// TwinCAT 3 PLC project XtsTransport
// Title: XTS Transport
// Author: D.Hauer
// ProjectVersion: 0.0.1
// Description: basic functionblocks for building XTS transport
// ProgramVersion: 3.1.4024.0
// libraries:
//   Tc2_Math, * (Beckhoff Automation GmbH)
//   Tc2_MC2, * (Beckhoff Automation GmbH)
//   Tc2_Standard, * (Beckhoff Automation GmbH)
//   Tc2_System, * (Beckhoff Automation GmbH)
//   Tc2_Utilities, * (Beckhoff Automation GmbH)
//   Tc3_McCollisionAvoidance, * (Beckhoff Automation GmbH)
//   Tc3_McCoordinatedMotion, * (Beckhoff Automation GmbH)
//   Tc3_Module, * (Beckhoff Automation GmbH)
//   Tc3_XTS_Utility, * (Beckhoff Automation GmbH)
//   VisuDialogs, * (System)
// project tree:
//   DUTs/_Visu/ ST_VisuExampleIO.TcDUT
//   / GlobalTextList.TcGTLO (not stored), MAIN.TcPOU (not stored), PlcTask.TcTTO (not stored), Visualization Manager.TcVMO (not stored)
//   POUs/ FB_OperatingMode.TcPOU, FB_SimpleCaExample.TcPOU (not stored)
//   VISUs/ CA_Visu.TcVIS
//   VISUs/Frame/ FrameVisuSimpelCaExample.TcVIS
//   VISUs/Frame/SubFrame/ FrameAdvancedMotion.TcVIS, FrameDummy.TcVIS, FrameXtsStateModel.TcVIS, FrameDislaimer.TcVIS
//   XTS/CaGroup/ FB_CaGroup.TcPOU, I_CaGroup.TcIO (not stored)
//   XTS/CaGroup/old/ fb_CaGroup_withOutInterface.TcPOU (not stored), fb_GroupCtrl.TcPOU
//   XTS/CaGroup/types/ E_GROUP_CHECK.TcDUT (not stored), E_GROUP_CTRL.TcDUT, E_GROUP_STATE.TcDUT, ST_GROUP_CTRL.TcDUT (not stored), ST_GROUP_INFO.TcDUT (not stored), ST_GROUP_STATE.TcDUT
//   XTS/ GVL_XTS.TcGVL (not stored), Param.TcGVL
//   XTS/Mover/ fb_Mover.TcPOU (not stored), I_Mover.TcIO, I_StationMover.TcIO
//   XTS/Mover/old/ fb_MoverCtrl.TcPOU (not stored), fb_Mover_withOutInterface.TcPOU (not stored)
//   XTS/Mover/types/ E_MOVER_CTRL.TcDUT (not stored), E_MOVER_STATE.TcDUT (not stored), ST_GEAR_DATA.TcDUT (not stored), ST_MOVER_CTRL.TcDUT (not stored), ST_MOVER_INFO.TcDUT (not stored), ST_MOVER_STATE.TcDUT (not stored), ST_MOVE_DATA.TcDUT (not stored)
//   XTS/Station/ fb_Station.TcPOU (not stored)
//   XTS/Station/types/ E_STATION_CTRL.TcDUT (not stored), E_STATION_STATE.TcDUT, fb_Station_LinkedListCtrl.TcPOU (not stored), I_Station_LinkedList.TcIO, ST_STATION_CTRL.TcDUT (not stored), ST_STATION_LIST_RESULT.TcDUT (not stored), ST_STATION_MOVER_DATA.TcDUT, ST_STATION_PARAMETER.TcDUT (not stored), ST_STATION_STATE.TcDUT, T_NEST_OFFSET.TcDUT
//   XTS/_types/ E_OperatingState.TcDUT (not stored), E_OperatingCmd.TcDUT (not stored), E_PROGRESS.TcDUT (not stored)

// ---- DUTs/_Visu/ST_VisuExampleIO.TcDUT
TYPE ST_VisuExampleIO :
STRUCT
	
	bStart				: BOOL;
	iState				: INT;
	bAgain				: BOOL := TRUE;
	fSetPos1			: LREAL := 1000;
	fSetPos2			: LREAL := 1250;
	fSetPos3			: LREAL := 1990;

	bStepModeActive		: BOOL;
	bNextStep			: BOOL;
	
// Operatin State
	eOPMState			: E_OperatingState;
	eLastOPMState		: E_OperatingState;
	eStateCommand		: E_OperatingCmd;
	
// CaGroup State
	stCaGroup			: REFERENCE TO AXES_GROUP_REF;	
	
END_STRUCT
END_TYPE

// ---- XTS/CaGroup/types/E_GROUP_CTRL.TcDUT
{attribute 'qualified_only'}
{attribute 'strict'}
{attribute 'to_string'}
TYPE E_GROUP_CTRL :
(
  GROUP_INVALID,
  GROUP_INIT    := 10,
  GROUP_CLEAR,
  GROUP_BUILD,
  GROUP_ENABLE
)UINT;
END_TYPE

// ---- XTS/CaGroup/types/E_GROUP_STATE.TcDUT
{attribute 'qualified_only'}
{attribute 'to_string'}
TYPE E_GROUP_STATE :
(
  GROUP_INVALID,
  GROUP_INIT    := 10,
  GROUP_CLEAR,
  GROUP_BUILD,
  GROUP_ENABLE

)UINT;
END_TYPE

// ---- XTS/CaGroup/types/ST_GROUP_STATE.TcDUT
TYPE ST_GROUP_STATE :
STRUCT
  State           : E_GROUP_STATE;
  McState         : MC_GROUP_STATE;
  AxisCount       : UINT;
END_STRUCT
END_TYPE

// ---- XTS/Station/types/E_STATION_STATE.TcDUT
{attribute 'to_string'}
TYPE E_STATION_STATE :
(
	STATION_NO_INIT,                // startup state after power on
  STATION_INIT,                   // station and list/queue cleared;
  STATION_DISABLE         := 10,  // check enable from ctrl
  STATION_ENABLE,                 // check enable from ctrl
  STATION_DETECT_MOVER,           // wait until queue > 0
  STATION_MOVER_ENTER     := 20,  // mover asking for entry
  STATION_MOVER_IN_TARGET,        // mover moving to PosWork
  STATION_PROCESS_START   := 30,  // wait until process started
  STATION_PROCESS_DONE,           // wait until process done
  STATION_CHECK           := 40,  // check for next nest in mask
  STATION_CHECK_NEST,             // get next nest position
  STATION_MOVER_OUT       := 50,  // mover asking to leave
  STATION_MOVER_RELEASE,          // check if release distance is passed
  STATION_MOVER_GONE,             // mover out of station, enter mover in target station list


  STATION_ERROR           := 127,
  STATION_ERROR_LIST_GET_HEAD_FAULT,
  STATION_ERROR_LIST_REMOVE_HEAD_FAULT,
  STATION_ERROR_LIST_ADD_TAIL_FAULT,
  STATION_ERROR_LIST_STATION_ID_WRONG,
  STATION_ERROR_LIST_MOVER_ID_INVALID,
  STATION_ERROR_INFEED_ERROR,
  STATION_ERROR_OUTFEED_TARGET_INVALID,

  STATION_ERROR_FATAL     := 255 // the thing that must not be
)USINT;
END_TYPE

// ---- XTS/Station/types/ST_STATION_MOVER_DATA.TcDUT
{attribute 'pack_mode' := '2'}
TYPE ST_STATION_MOVER_DATA :
STRUCT
  nMoverId        : USINT;  // who am I?  !! MUST be correct !! - movement to base position sets everything in order, DO NOT manipulate!
  nTargetStation  : USINT;  // where shall I be? used for double checking with StationId at infeed of mover into station

  {attribute 'displaymode':='bin'}
  nMask           : BYTE;   // how many of you are there? (1 = default, no action required)

  rOffset         : REAL;   // offset for use in work flow !! added to static mover offset for every nest(bit) in nMask!!
END_STRUCT
END_TYPE

// ---- XTS/Station/types/ST_STATION_STATE.TcDUT
{attribute 'pack_mode' := '2'}
TYPE ST_STATION_STATE :
STRUCT
  eState          : E_STATION_STATE;
  {attribute 'displaymode':='bin'}
  nMask           : BYTE;
  nMoverId        : USINT;
  nQueue          : USINT; // queue count for station
END_STRUCT
END_TYPE

// ---- XTS/Station/types/T_NEST_OFFSET.TcDUT
TYPE T_NEST_OFFSET : ARRAY[1..MAX_MOVER]        OF
                     ARRAY[1..MAX_STATION_POS]  OF LREAL;
END_TYPE

// ---- XTS/Param.TcGVL
//{attribute 'qualified_only'}
VAR_GLOBAL CONSTANT
// HAUD 2023 12 13
  Version             : STRING  := '3.2.0'; // V3.2.0 - design test with references, improved separation of Mover and Group handling, redesign of group handling



// XTS-Constant ´--> using Tc3_XTS_Utility.TcIoXtsEnvironmentParameterList


  MAX_INFO_SERVER     : UINT    :=  TO_UINT(Tc3_XTS_Utility.TcIoXtsEnvironmentParameterList.MaxXtsInfoServer);
  MAX_INFO_STATION    : UINT    :=  TO_UINT(Tc3_XTS_Utility.TcIoXtsEnvironmentParameterList.MaxXtsInfoStation);
  MAX_INFO_STOP_POS   : UINT    :=  TO_UINT(Tc3_XTS_Utility.TcIoXtsEnvironmentParameterList.MaxXtsStopPositionsPerStation);


  MAX_MOVER           : UINT    := TO_UINT(Tc3_XTS_Utility.TcIoXtsEnvironmentParameterList.MaxXtsMoversPerXpu);
  MAX_MODULE          : UINT    := TO_UINT(Tc3_XTS_Utility.TcIoXtsEnvironmentParameterList.MaxModulesPerPart);
  MAX_PART            : UINT    := TO_UINT(Tc3_XTS_Utility.TcIoXtsEnvironmentParameterList.MaxXtsPartsPerXpu);
  MAX_TRACK           : UINT    := TO_UINT(Tc3_XTS_Utility.TcIoXtsEnvironmentParameterList.MaxXtsTracksPerXpu);
  MAX_GROUP           : UINT    := TO_UINT(Tc3_XTS_Utility.TcIoXtsEnvironmentParameterList.MaxXtsCaGroup);

  MAX_STATION         : UINT    := 2;
  MAX_STATION_POS     : UINT    := TO_UINT(SIZEOF(ST_STATION_STATE.nMask)*8);
  MAX_LIST_NODES      : UINT    := MAX_MOVER;
  MAX_MASTER          : UINT    := 1;
  
END_VAR

// ---- XTS/Mover/I_Mover.TcIO
INTERFACE I_Mover

METHOD Disable : E_PROGRESS
VAR_INPUT
  Execute             : BOOL;
END_VAR
END_METHOD

METHOD Enable : E_PROGRESS
VAR_INPUT
  Execute             : BOOL;
END_VAR
END_METHOD

METHOD GearIn : E_PROGRESS;
VAR_INPUT
  Execute             : BOOL;
  stGearData          : ST_GEAR_DATA;
  stMoveData          : ST_MOVE_DATA;
END_VAR
END_METHOD

METHOD GearInPosCa : E_PROGRESS
VAR_INPUT
  Execute             : BOOL;
  stMoveData          : ST_MOVE_DATA;
  stGearData          : ST_GEAR_DATA;  
END_VAR
END_METHOD

METHOD GearOut : E_PROGRESS
VAR_INPUT
  Execute             : BOOL;
END_VAR
END_METHOD

METHOD GetMoverInfo : ST_MOVER_INFO
VAR_INPUT
END_VAR
END_METHOD

METHOD Halt : E_PROGRESS
VAR_INPUT
  Execute             : BOOL;
  stMoveData          : ST_MOVE_DATA;
END_VAR
END_METHOD

PROPERTY LastGap : REFERENCE to lreal
SET
END_SET
END_PROPERTY

PROPERTY LastPosition : REFERENCE to LREAL
SET
END_SET
END_PROPERTY

PROPERTY Master : REFERENCE to AXIS_REF
SET
END_SET
END_PROPERTY

PROPERTY Mover : REFERENCE to AXIS_REF
SET
END_SET
END_PROPERTY

METHOD MoveToPosCa : E_PROGRESS
VAR_INPUT
  Execute             : BOOL;
  stMoveData          : ST_MOVE_DATA;
END_VAR
END_METHOD

PROPERTY RailLength : LREAL
GET
END_GET
SET
END_SET
END_PROPERTY

METHOD Reset : E_PROGRESS
VAR_INPUT
  Execute             : BOOL;
END_VAR
END_METHOD

METHOD SendToPosCa : E_PROGRESS
VAR_INPUT
  Execute             : BOOL;
  stMoveData          : ST_MOVE_DATA;
END_VAR
END_METHOD

END_INTERFACE

// ---- XTS/Mover/I_StationMover.TcIO
INTERFACE I_StationMover

METHOD GetMoverInfo : ST_MOVER_INFO
VAR_INPUT
END_VAR
END_METHOD

METHOD MoveToPosCa : E_PROGRESS
VAR_INPUT
  Execute             : BOOL;
  stMoveData          : ST_MOVE_DATA;
END_VAR
END_METHOD

PROPERTY RailLength : LREAL
GET
END_GET
END_PROPERTY

METHOD SendToPosCa : E_PROGRESS
VAR_INPUT
  Execute             : BOOL;
  stMoveData          : ST_MOVE_DATA;
END_VAR
END_METHOD

END_INTERFACE

// ---- XTS/Station/types/I_Station_LinkedList.TcIO
INTERFACE I_Station_LinkedList

METHOD AddHeadValue : ST_STATION_LIST_RESULT
VAR_INPUT
  stData        : ST_STATION_MOVER_DATA;
END_VAR
END_METHOD

METHOD AddTailValue : ST_STATION_LIST_RESULT
VAR_INPUT
  stData          : ST_STATION_MOVER_DATA;
END_VAR
END_METHOD

PROPERTY Count : UDINT
GET
END_GET
END_PROPERTY

PROPERTY Data : ARRAY[0..MAX_LIST_NODES] OF ST_STATION_MOVER_DATA
GET
END_GET
END_PROPERTY

PROPERTY Free : UDINT
GET
END_GET
END_PROPERTY

METHOD GetHead : ST_STATION_LIST_RESULT
VAR_INPUT
END_VAR
END_METHOD

METHOD InitList : BOOL
END_METHOD

PROPERTY Nodes : ARRAY[0..MAX_LIST_NODES] OF T_LinkedListEntry
GET
END_GET
END_PROPERTY

METHOD RemoveHeadValue : ST_STATION_LIST_RESULT
VAR_INPUT
END_VAR
END_METHOD

END_INTERFACE

// ---- POUs/FB_OperatingMode.TcPOU
FUNCTION_BLOCK FB_OperatingMode
//---------------------------------------------------------------------------------------------------------------
//
//  Fen 2023.12.21
//
//  - XTS_TRAINING
//  - example project for setting up transport layer
//
//
//  FB_OperatingMode
//  - Operating Mode handler for XTS_training Exsample
//  - 
//
//
//---------------------------------------------------------------------------------------------------------------
// This SOFTWARE is provided as an Exemple by THE PROVIDER "as is" and "with all faults." THE PROVIDER makes no 
// representations or warranties of any kind concerning the safety, suitability, lack of viruses, inaccuracies, 
// typographical errors, or other harmful components of this SOFTWARE. There are inherent dangers in the use of 
// any software, and you are solely responsible for determining whether this SOFTWARE is compatible with your 
// equipment and other software installed on your equipment. You are also solely responsible for the protection 
// of your equipment and backup of your data, and THE PROVIDER will not be liable for any damages you may suffer 
// in connection with using, modifying, or distributing this SOFTWARE.
//---------------------------------------------------------------------------------------------------------------

VAR 
	_eState			: E_OperatingState;	
	_eLastState		: E_OperatingState;

	_eCommand		: E_OperatingCmd;
	_eActCommand	: E_OperatingCmd;
	

	_StaeCompleteRtrig	:R_TRIG;
	_StaeComplete		: BOOL;

	
	_bSingelStep				: BOOL;

END_VAR

PROPERTY Command : E_OperatingCmd
GET

	Command := _eActCommand;
END_GET
SET

	_eCommand := Command;
END_SET
END_PROPERTY

METHOD Cyclic
VAR_INPUT
END_VAR
// simple Example for Operatingmode handler


// State Complete
	_StaeCompleteRtrig();
	IF _StaeCompleteRtrig.Q THEN
		_StaeComplete := TRUE;
	END_IF

// Xts Operating Mode

	_eActCommand := _eActCommand;

	CASE _eState OF
	
	// Invalid 	--> wait for Cmd 	
	E_OperatingState.OperatingMode_INVALID : 
		IF _eCommand = E_OperatingCmd.OperatingCmd_Clear THEN
			_eState := E_OperatingState.OperatingMode_Clear;
			_eActCommand := E_OperatingCmd.OperatingCmd_DONE;
			_eLastState := E_OperatingState.OperatingMode_INVALID;
		
		ELSE 
			_eActCommand := E_OperatingCmd.OperatingCmd_DONE;	
		END_IF
		
	// Clear 	--> Init Ca-Group  and Axis 	
	E_OperatingState.OperatingMode_Clear:
		IF _StaeComplete 
		THEN
			_StaeComplete := FALSE;
			_eState := E_OperatingState.OperatingMode_Clear_Sc;
		END_IF
		
		CASE _eCommand	OF  			
			E_OperatingCmd.OperatingCmd_Reset :	
				_eState := E_OperatingState.OperatingMode_Reset;
				_eActCommand := E_OperatingCmd.OperatingCmd_DONE;
				_eLastState := E_OperatingState.OperatingMode_Clear;
			
		ELSE 
			_eActCommand := E_OperatingCmd.OperatingCmd_DONE;	
				
		END_CASE
		
	// Clear_Sc 	--> State complete	
	E_OperatingState.OperatingMode_Clear_Sc :
		CASE _eCommand	OF  
			E_OperatingCmd.OperatingCmd_Clear :
				_eState := E_OperatingState.OperatingMode_Clear;
				_eActCommand := E_OperatingCmd.OperatingCmd_DONE;
				_eLastState := E_OperatingState.OperatingMode_Clear_Sc;
			
			E_OperatingCmd.OperatingCmd_Reset :	
				_eState := E_OperatingState.OperatingMode_Reset;
				_eActCommand := E_OperatingCmd.OperatingCmd_DONE;
				_eLastState := E_OperatingState.OperatingMode_Clear_Sc;
				
			E_OperatingCmd.OperatingCmd_Prepare	:
				_eState := E_OperatingState.OperatingMode_Prepare;
				_eActCommand := E_OperatingCmd.OperatingCmd_DONE;
				_eLastState := E_OperatingState.OperatingMode_Clear_Sc;
		
		ELSE 
			_eActCommand := E_OperatingCmd.OperatingCmd_DONE;	
				
		END_CASE
		
	
	// Prepare 	--> build Ca-Group  and enable Axis 	
	E_OperatingState.OperatingMode_Prepare :
		IF _StaeComplete 
		THEN
			_StaeComplete := FALSE;
			_eState := E_OperatingState.OperatingMode_Prepar_Sc;
		END_IF
		
		CASE _eCommand	OF  
			E_OperatingCmd.OperatingCmd_Clear :
				_eState := E_OperatingState.OperatingMode_Clear;
				_eActCommand := E_OperatingCmd.OperatingCmd_DONE;
				_eLastState := E_OperatingState.OperatingMode_Prepare;
			
			E_OperatingCmd.OperatingCmd_Reset :	
				_eState := E_OperatingState.OperatingMode_Reset;
				_eActCommand := E_OperatingCmd.OperatingCmd_DONE;
				_eLastState := E_OperatingState.OperatingMode_Prepare;
		
		ELSE 
			_eActCommand := E_OperatingCmd.OperatingCmd_DONE;	
		END_CASE
	
	// Stopping 	--> stop Axis 		
	E_OperatingState.OperatingMode_Stopping :
		IF _StaeComplete 
		THEN
			_StaeComplete := FALSE;
			_eState := E_OperatingState.OperatingMode_Prepar_Sc;
		END_IF
		CASE _eCommand	OF  
			E_OperatingCmd.OperatingCmd_Clear :
				_eState := E_OperatingState.OperatingMode_Clear;
				_eActCommand := E_OperatingCmd.OperatingCmd_DONE;
				_eLastState := E_OperatingState.OperatingMode_Stopping;
			
			E_OperatingCmd.OperatingCmd_Reset :	
				_eState := E_OperatingState.OperatingMode_Reset;
				_eActCommand := E_OperatingCmd.OperatingCmd_DONE;
				_eLastState := E_OperatingState.OperatingMode_Stopping;
		
		ELSE 
			_eActCommand := E_OperatingCmd.OperatingCmd_DONE;	
		END_CASE
		
	// Prepare 	--> emptying the system 		
	E_OperatingState.OperatingMode_Empty:
		IF _StaeComplete 
		THEN
			_StaeComplete := FALSE;
			_eState := E_OperatingState.OperatingMode_Prepar_Sc;
		END_IF
		
		CASE _eCommand	OF  
			E_OperatingCmd.OperatingCmd_Clear :
				_eState := E_OperatingState.OperatingMode_Clear;
				_eActCommand := E_OperatingCmd.OperatingCmd_DONE;
				_eLastState := E_OperatingState.OperatingMode_Empty;
			
			E_OperatingCmd.OperatingCmd_Reset :	
				_eState := E_OperatingState.OperatingMode_Reset;
				_eActCommand := E_OperatingCmd.OperatingCmd_DONE;
				_eLastState := E_OperatingState.OperatingMode_Empty;
				
			E_OperatingCmd.OperatingCmd_Stopping :
				_eState := E_OperatingState.OperatingMode_Stopping;
				_eActCommand := E_OperatingCmd.OperatingCmd_DONE;
				_eLastState := E_OperatingState.OperatingMode_Empty;
		
		ELSE 
			_eActCommand := E_OperatingCmd.OperatingCmd_DONE;	
			
		END_CASE
	
	// 	Prepare 	--> State complete
	E_OperatingState.OperatingMode_Prepar_Sc:
		CASE _eCommand	OF  
			E_OperatingCmd.OperatingCmd_Clear :
				_eState := E_OperatingState.OperatingMode_Clear;
				_eActCommand := E_OperatingCmd.OperatingCmd_DONE;
				_eLastState := E_OperatingState.OperatingMode_Prepar_Sc;
			
			E_OperatingCmd.OperatingCmd_Reset :	
				_eState := E_OperatingState.OperatingMode_Reset;
				_eActCommand := E_OperatingCmd.OperatingCmd_DONE;
				_eLastState := E_OperatingState.OperatingMode_Prepar_Sc;
				
			E_OperatingCmd.OperatingCmd_Stopping :
				_eState := E_OperatingState.OperatingMode_Stopping;
				_eActCommand := E_OperatingCmd.OperatingCmd_DONE;
				_eLastState := E_OperatingState.OperatingMode_Prepar_Sc;
			
			E_OperatingCmd.OperatingCmd_Home 	:
				_eState := E_OperatingState.OperatingMode_Home;
				_eActCommand := E_OperatingCmd.OperatingCmd_DONE;
				_eLastState := E_OperatingState.OperatingMode_Prepar_Sc;
		
		ELSE 
			_eActCommand := E_OperatingCmd.OperatingCmd_DONE;	
	
		END_CASE
		
	// 	Empty 	--> State complete
	E_OperatingState.OperatingMode_Empty_Sc:
			_eState := E_OperatingState.OperatingMode_Prepar_Sc;
			_eLastState := E_OperatingState.OperatingMode_Empty_Sc;
		
	// 	Stopping 	--> State complete
	E_OperatingState.OperatingMode_Stopping_Sc:
			_eState := E_OperatingState.OperatingMode_Prepar_Sc;
			_eLastState := E_OperatingState.OperatingMode_Stopping_Sc;


	
	// 	Home 	--> Move to Start Position
	E_OperatingState.OperatingMode_Home :
		IF _StaeComplete 
		THEN
			_StaeComplete := FALSE;
			_eState := E_OperatingState.OperatingMode_Home_Sc;
		END_IF
		
		CASE _eCommand	OF  
			E_OperatingCmd.OperatingCmd_Clear :
				_eState := E_OperatingState.OperatingMode_Clear;
				_eActCommand := E_OperatingCmd.OperatingCmd_DONE;
				_eLastState := E_OperatingState.OperatingMode_Home;
			
			E_OperatingCmd.OperatingCmd_Reset :	
				_eState := E_OperatingState.OperatingMode_Reset;
				_eActCommand := E_OperatingCmd.OperatingCmd_DONE;
				_eLastState := E_OperatingState.OperatingMode_Home;
				
			E_OperatingCmd.OperatingCmd_Stopping :
				_eState := E_OperatingState.OperatingMode_Stopping;
				_eActCommand := E_OperatingCmd.OperatingCmd_DONE;
				_eLastState := E_OperatingState.OperatingMode_Home;
		
		ELSE 
			_eActCommand := E_OperatingCmd.OperatingCmd_DONE;	
	
		END_CASE
	
	// 	Home 	--> State complete
	E_OperatingState.OperatingMode_Home_Sc :	
		_eState := E_OperatingState.OperatingMode_Active;
		
		CASE _eCommand	OF  
			E_OperatingCmd.OperatingCmd_Clear :
				_eState := E_OperatingState.OperatingMode_Clear;
				_eActCommand := E_OperatingCmd.OperatingCmd_DONE;
				_eLastState := E_OperatingState.OperatingMode_Home_Sc;
			
			E_OperatingCmd.OperatingCmd_Reset :	
				_eState := E_OperatingState.OperatingMode_Reset;
				_eActCommand := E_OperatingCmd.OperatingCmd_DONE;
				_eLastState := E_OperatingState.OperatingMode_Home_Sc;
				
			E_OperatingCmd.OperatingCmd_Stopping :
				_eState := E_OperatingState.OperatingMode_Stopping;
				_eActCommand := E_OperatingCmd.OperatingCmd_DONE;
				_eLastState := E_OperatingState.OperatingMode_Home_Sc;
		
		ELSE 
			_eActCommand := E_OperatingCmd.OperatingCmd_DONE;	
	
		END_CASE
	
	// 	Active/Work 	--> execute work sequences
 	E_OperatingState.OperatingMode_Active :
		CASE _eCommand	OF  
			E_OperatingCmd.OperatingCmd_Clear :
				_eState := E_OperatingState.OperatingMode_Clear;
				_eActCommand := E_OperatingCmd.OperatingCmd_DONE;
				_eLastState := E_OperatingState.OperatingMode_Active;
			
			E_OperatingCmd.OperatingCmd_Reset :	
				_eState := E_OperatingState.OperatingMode_Reset;
				_eActCommand := E_OperatingCmd.OperatingCmd_DONE;
				_eLastState := E_OperatingState.OperatingMode_Active;
				
			E_OperatingCmd.OperatingCmd_Stopping :
				_eState := E_OperatingState.OperatingMode_Stopping;
				_eActCommand := E_OperatingCmd.OperatingCmd_DONE;
				_eLastState := E_OperatingState.OperatingMode_Active;
			
			E_OperatingCmd.OperatingCmd_Empty 	:
				_eState := E_OperatingState.OperatingMode_Empty;
				_eActCommand := E_OperatingCmd.OperatingCmd_DONE;
				_eLastState := E_OperatingState.OperatingMode_Active;
		
		ELSE 
			_eActCommand := E_OperatingCmd.OperatingCmd_DONE;	
				
		END_CASE
	
	// 	Reset 	--> Reset Error --> Jump to last state back
	E_OperatingState.OperatingMode_Reset :
		IF _StaeComplete 
		THEN
			_StaeComplete := FALSE;
			_eState := _eLastState;
			_eLastState := E_OperatingState.OperatingMode_Reset;
		END_IF
	
		_eActCommand := E_OperatingCmd.OperatingCmd_DONE;
		
	
	END_CASE
END_METHOD

PROPERTY eLastState : E_OperatingState
GET

	eLastState := _eLastState;
END_GET
END_PROPERTY

PROPERTY eState : E_OperatingState
GET

	eState := _eState;
END_GET
END_PROPERTY

METHOD M_StateComplete
VAR_INPUT
END_VAR

	//_StaeCompleteRtrig.CLK := TRUE;
	_StaeComplete := TRUE;
END_METHOD

PROPERTY sState : STRING
GET

	sState := to_String(_eState);
END_GET
END_PROPERTY

END_FUNCTION_BLOCK

// ---- XTS/CaGroup/FB_CaGroup.TcPOU
//---------------------------------------------------------------------------------------------------------------
//
//  HAUD 2023.12.13
//
//
//  fb_CaGroup
//  - handles CA group states
//  - add mover to group
//  - remove mover from group
//  - clear group error
//  - startup procedure for getting group ready to work
//
//
//  VAR INPUT / OUTPUT --> see properties
//
//---------------------------------------------------------------------------------------------------------------//
// This SOFTWARE is provided as an Exemple by THE PROVIDER "as is" and "with all faults." THE PROVIDER makes no  //
// representations or warranties of any kind concerning the safety, suitability, lack of viruses, inaccuracies,  //
// typographical errors, or other harmful components of this SOFTWARE. There are inherent dangers in the use of  //
// any software, and you are solely responsible for determining whether this SOFTWARE is compatible with your    //
// equipment and other software installed on your equipment. You are also solely responsible for the protection  //
// of your equipment and backup of your data, and THE PROVIDER will not be liable for any damages you may suffer //
// in connection with using, modifying, or distributing this SOFTWARE.                                           //
//---------------------------------------------------------------------------------------------------------------//
FUNCTION_BLOCK FB_CaGroup	IMPLEMENTS I_CaGroup
VAR
  _eCheck                     : E_GROUP_CHECK;
  _bError                     : BOOL;

  _GroupRef                   : REFERENCE TO Tc3_McCoordinatedMotion.AXES_GROUP_REF;
  _GroupCommon                : MCTOPLC_GROUP_COMMON_PART;

  _AxisRefMover               : REFERENCE TO ARRAY[1..MAX_MOVER] OF Tc2_MC2.AXIS_REF;


  // MC2 function block for halting all motion commands on mover before switching off group
  _fbHalt                     : ARRAY[1..MAX_MOVER] OF Tc2_MC2.MC_Halt;
  _fbReset                    : ARRAY[1..MAX_MOVER] OF Tc2_MC2.MC_Reset;

  // CA group fb instances
  _fbAddAxisGroup             : ARRAY[1..MAX_MOVER] OF Tc3_McCoordinatedMotion.MC_AddAxisToGroup;
  _fbRemoveAxisGroup          : ARRAY[1..MAX_MOVER] OF Tc3_McCoordinatedMotion.MC_RemoveAxisFromGroup;

  _fbGroupDisable             : Tc3_McCoordinatedMotion.MC_GroupDisable;
  _fbGroupEnable              : Tc3_McCoordinatedMotion.MC_GroupEnable;
  _fbGroupErrorRead           : Tc3_McCoordinatedMotion.MC_GroupReadError;
  _fbGroupStatusRead          : Tc3_McCoordinatedMotion.MC_GroupReadStatus;
  _fbGroupReset               : Tc3_McCoordinatedMotion.MC_GroupReset;

  _stGroupInfo                : ST_GROUP_INFO;  // additional bits about the state of the CA group

  _rtrigGroupStatusRead,
  _rtrigGroupErrorRead        : Tc2_Standard.R_TRIG;


END_VAR

METHOD AddAll : E_PROGRESS
VAR_INPUT
  Execute     : BOOL;
END_VAR
VAR_INST
  _nErrorId   : UDINT;
  _eState     : E_PROGRESS;

  _nMover     : UINT;
END_VAR
IF NOT Execute THEN _eState     := E_PROGRESS.PROGRESS_INIT; END_IF 
IF NOT Check() THEN AddAll := E_PROGRESS.PROGRESS_ERROR; RETURN; END_IF


CASE _eState
OF
  E_PROGRESS.PROGRESS_INIT:
    IF Execute
    THEN
      _nErrorId               := 0;
      _nMover                 := 1;
      _eState                 := E_PROGRESS.PROGRESS_BUSY;
    END_IF
END_CASE
//-----------------------------------------------------------------------------
//-----------------------------------------------------------------------------
CASE _eState
OF
  E_PROGRESS.PROGRESS_BUSY:
    _eState                   := E_PROGRESS.PROGRESS_PREPARE;
    _fbAddAxisGroup[_nMover](
                AxesGroup     := _GroupRef, 
                Axis          := _AxisRefMover[_nMover], 
                Execute       := FALSE, 
                IdentInGroup  := UDINT_TO_IDENTINGROUP(_AxisRefMover[_nMover].NcToPlc.AxisId));
END_CASE
//-----------------------------------------------------------------------------
//-----------------------------------------------------------------------------
CASE _eState
OF
  E_PROGRESS.PROGRESS_PREPARE:
    _fbAddAxisGroup[_nMover](
                AxesGroup     := _GroupRef, 
                Axis          := _AxisRefMover[_nMover], 
                Execute       := TRUE, 
                IdentInGroup  := UDINT_TO_IDENTINGROUP(_AxisRefMover[_nMover].NcToPlc.AxisId));

    IF (_fbAddAxisGroup[_nMover].Error)
    THEN
      _eState                 := E_PROGRESS.PROGRESS_ERROR;
      _nErrorId               := _fbAddAxisGroup[_nMover].ErrorId;

    ELSIF (_fbAddAxisGroup[_nMover].Done)
    THEN
      _eState                 := E_PROGRESS.PROGRESS_CHECK;
    END_IF
END_CASE
//-----------------------------------------------------------------------------
//-----------------------------------------------------------------------------
CASE _eState
OF
  E_PROGRESS.PROGRESS_CHECK:
    _eState                   := E_PROGRESS.PROGRESS_OCCUPIED;
    _fbAddAxisGroup[_nMover](
                AxesGroup     := _GroupRef, 
                Axis          := _AxisRefMover[_nMover], 
                Execute       := FALSE, 
                IdentInGroup  := UDINT_TO_IDENTINGROUP(_AxisRefMover[_nMover].NcToPlc.AxisId));
END_CASE
//-----------------------------------------------------------------------------
//-----------------------------------------------------------------------------
CASE _eState
OF
  E_PROGRESS.PROGRESS_OCCUPIED:
    _nMover                   := _nMover + 1;

    IF NOT (_nMover > MAX_MOVER)
    THEN
      _eState                 := E_PROGRESS.PROGRESS_BUSY;
    ELSE
      _eState                 := E_PROGRESS.PROGRESS_DONE;
    END_IF
END_CASE
//-----------------------------------------------------------------------------
//-----------------------------------------------------------------------------

AddAll                   := _eState;
END_METHOD

PROPERTY AxisRef : REFERENCE TO ARRAY[1..MAX_MOVER] OF Tc2_MC2.AXIS_REF
SET
_AxisRefMover REF= AxisRef;
END_SET
END_PROPERTY

METHOD PROTECTED Check : BOOL

IF NOT __ISVALIDREF(_GroupRef)
THEN
  _eCheck                     := E_GROUP_CHECK.CHECK_GROUP_REF_INVALID;
  RETURN;
END_IF

IF NOT __ISVALIDREF(_AxisRefMover)
THEN
  _eCheck                     := E_GROUP_CHECK.CHECK_AXIS_REF_INVALID;
  RETURN;
END_IF

_eCheck                       := E_GROUP_CHECK.CHECK_DONE;
Check                         := TRUE;
END_METHOD

METHOD Disable : E_PROGRESS
VAR_INPUT
  Execute     : BOOL;
END_VAR
VAR_INST
  _nErrorId   : UDINT;
  _eState     : E_PROGRESS;

  _nMover     : UINT;
END_VAR
IF NOT Execute THEN _eState       := E_PROGRESS.PROGRESS_INIT; END_IF 
IF NOT Check() THEN Disable  := E_PROGRESS.PROGRESS_ERROR; RETURN; END_IF


CASE _eState
OF
  E_PROGRESS.PROGRESS_INIT:
    IF Execute
    THEN
      _nErrorId               := 0;
      _nMover                 := 1;
      _eState                 := E_PROGRESS.PROGRESS_BUSY;
    END_IF
END_CASE
//-----------------------------------------------------------------------------
//-----------------------------------------------------------------------------
CASE _eState
OF
  E_PROGRESS.PROGRESS_BUSY:
    _eState                   := E_PROGRESS.PROGRESS_PREPARE;
    _fbGroupDisable(
              AxesGroup       := _GroupRef, 
              Execute         := FALSE); 
END_CASE
//-----------------------------------------------------------------------------
//-----------------------------------------------------------------------------
CASE _eState
OF
  E_PROGRESS.PROGRESS_PREPARE:
    _fbGroupDisable(
              AxesGroup       := _GroupRef, 
              Execute         := TRUE); 

    IF (_fbGroupDisable.Error)
    THEN
      _eState                 := E_PROGRESS.PROGRESS_ERROR;
      _nErrorId               := _fbGroupDisable.ErrorId;
      _fbGroupDisable(
              AxesGroup       := _GroupRef, 
              Execute         := FALSE); 


    ELSIF (_fbGroupDisable.Done)
    THEN
      _eState                 := E_PROGRESS.PROGRESS_DONE;
      _fbGroupDisable(
              AxesGroup       := _GroupRef, 
              Execute         := FALSE); 
    END_IF
END_CASE
//-----------------------------------------------------------------------------
//-----------------------------------------------------------------------------

Disable                  := _eState;
END_METHOD

METHOD Enable : E_PROGRESS
VAR_INPUT
  Execute     : BOOL;
END_VAR
VAR_INST
  _nErrorId   : UDINT;
  _eState     : E_PROGRESS;

  _nMover     : UINT;
END_VAR
IF NOT Execute THEN _eState       := E_PROGRESS.PROGRESS_INIT; END_IF 
IF NOT Check() THEN Enable   := E_PROGRESS.PROGRESS_ERROR; RETURN; END_IF


CASE _eState
OF
  E_PROGRESS.PROGRESS_INIT:
    IF Execute
    THEN
      _nErrorId               := 0;
      _nMover                 := 1;
      _eState                 := E_PROGRESS.PROGRESS_BUSY;
    END_IF
END_CASE
//-----------------------------------------------------------------------------
//-----------------------------------------------------------------------------
CASE _eState
OF
  E_PROGRESS.PROGRESS_BUSY:
    _eState                   := E_PROGRESS.PROGRESS_PREPARE;
    _fbGroupEnable(
                AxesGroup     := _GroupRef, 
                Execute       := FALSE);
END_CASE
//-----------------------------------------------------------------------------
//-----------------------------------------------------------------------------
CASE _eState
OF
  E_PROGRESS.PROGRESS_PREPARE:
    _fbGroupEnable(
                AxesGroup     := _GroupRef, 
                Execute       := TRUE);

    IF (_fbGroupEnable.Error)
    THEN
      _eState                 := E_PROGRESS.PROGRESS_ERROR;
      _nErrorId               := _fbGroupEnable.ErrorId;

      _fbGroupEnable(
                AxesGroup     := _GroupRef, 
                Execute       := FALSE);

    ELSIF (_fbGroupEnable.Done)
    THEN
      _eState                 := E_PROGRESS.PROGRESS_DONE;

      _fbGroupEnable(
                AxesGroup     := _GroupRef, 
                Execute       := FALSE);
    END_IF
END_CASE
//-----------------------------------------------------------------------------
//-----------------------------------------------------------------------------

Enable                   := _eState;
END_METHOD

PROPERTY GroupInfo : reference to ST_GROUP_INFO
GET
GroupInfo REF= _stGroupInfo;
END_GET
END_PROPERTY

PROPERTY GroupRef : reference to Tc3_McCoordinatedMotion.AXES_GROUP_REF
GET
GroupRef REF= _GroupRef;
END_GET
SET
_GroupRef REF= GroupRef;
END_SET
END_PROPERTY

METHOD InfoCycle : DWORD
VAR_INPUT
  Enable          : BOOL;
END_VAR
VAR_INST
  _nErrorIdADS,
  _nErrorIdRead   : UDINT;
END_VAR
IF NOT Check() THEN RETURN; END_IF


//-----------------------------------------------------------------------------------------------
// cyclic CA group
//-----------------------------------------------------------------------------------------------
_fbGroupStatusRead(
              AxesGroup                     := _GroupRef, 
              Enable                        := Enable, 
              Valid                         => _stGroupInfo.GroupStatusValid, 
              Busy                          => _stGroupInfo.GroupStatusBusy, 
              GroupMoving                   => _stGroupInfo.GroupMoving, 
              GroupHoming                   => _stGroupInfo.GroupHoming, 
              GroupErrorStop                => _stGroupInfo.GroupErrorStop, 
              GroupNotReady                 => _stGroupInfo.GroupNotReady, 
              GroupStandby                  => _stGroupInfo.GroupStandby, 
              GroupStopping                 => _stGroupInfo.GroupStopping, 
              GroupDisabled                 => _stGroupInfo.GroupDisabled, 
              AllAxesStanding               => _stGroupInfo.AllAxesStanding, 
              ConstantVelocity              => _stGroupInfo.ConstantVelocity, 
              Accelerating                  => _stGroupInfo.Accelerating, 
              Decelerating                  => _stGroupInfo.Decelerating, 
              InPosition                    => _stGroupInfo.InPosition, 
              Error                         => , 
              ErrorId                       => );

_fbGroupErrorRead(
              AxesGroup                     := _GroupRef, 
              Enable                        := Enable, 
              ErrorId                       => , 
              GroupErrorId                  => );


_stGroupInfo.AxisCount := _GroupRef.NcToPlc.CA.Common.GroupAxesCount;		  
			  
// fetch group error
_rtrigGroupStatusRead(CLK                   := (_stGroupInfo.GroupError OR
                                                _stGroupInfo.GroupErrorStop));
IF _rtrigGroupStatusRead.Q
THEN
  _stGroupInfo.GroupError   := _bError      := TRUE;
  _stGroupInfo.GroupErrorId                 := _fbGroupErrorRead.GroupErrorId;
END_IF

// fetch internal fb error
_rtrigGroupErrorRead(CLK                    := _fbGroupErrorRead.Error);
IF _rtrigGroupErrorRead.Q
THEN
  _nErrorIdADS                              := _fbGroupErrorRead.ErrorId;
END_IF
END_METHOD

METHOD McHaltAll : E_PROGRESS
VAR_INPUT
  Execute       : BOOL;
END_VAR
VAR_INST
  _nErrorId     : UDINT;
  _eState       : E_PROGRESS;

  _nMover       : UINT;
END_VAR
IF NOT Execute 
THEN 
	_eState     := E_PROGRESS.PROGRESS_INIT; 
END_IF 
IF NOT Check() 
THEN 
	McHaltAll   := E_PROGRESS.PROGRESS_ERROR; 
	RETURN; 
END_IF


CASE _eState
OF
  E_PROGRESS.PROGRESS_INIT:
    IF Execute
    THEN
      _nErrorId               := 0;
      _nMover                 := 1;
      _eState                 := E_PROGRESS.PROGRESS_BUSY;
    END_IF
END_CASE

//-----------------------------------------------------------------------------
//-----------------------------------------------------------------------------
CASE _eState
OF
  E_PROGRESS.PROGRESS_BUSY:
    _eState                   := E_PROGRESS.PROGRESS_PREPARE;
    FOR _nMover := 1 TO MAX_MOVER
    DO
      _fbHalt[_nMover](
                Axis          := _AxisRefMover[_nMover], 
                Execute       := FALSE, 
                Deceleration  := 15_000, 
                Jerk          := 150_000, 
                BufferMode    := MC_BufferMode.MC_Aborting,
                Error=> , 
                ErrorID=> );
    END_FOR
END_CASE

//-----------------------------------------------------------------------------
//-----------------------------------------------------------------------------
CASE _eState
OF
  E_PROGRESS.PROGRESS_PREPARE:
    _GroupCommon              := _GroupRef.NcToPlc.Common;
    IF (_GroupCommon.GroupStatus.Flags.AllAxesStanding)
    THEN
      _eState                 := E_PROGRESS.PROGRESS_CHECK;
    END_IF

    FOR _nMover := 1 TO MAX_MOVER
    DO
      _fbHalt[_nMover](
                Axis          := _AxisRefMover[_nMover], 
                Execute       := TRUE, 
                Deceleration  := 15_000, 
                Jerk          := 150_000, 
                BufferMode    := MC_BufferMode.MC_Aborting,
                Error=> , 
                ErrorID=>);
      IF (_fbHalt[_nMover].Error)
      THEN
        _nErrorId             := _fbHalt[_nMover].ErrorID;
        _eState               := E_PROGRESS.PROGRESS_ERROR;
        EXIT;
      END_IF
    END_FOR
END_CASE

//-----------------------------------------------------------------------------
//-----------------------------------------------------------------------------
CASE _eState
OF
  E_PROGRESS.PROGRESS_CHECK:
    _eState                   := E_PROGRESS.PROGRESS_DONE;
    FOR _nMover := 1 TO MAX_MOVER
    DO
      _fbHalt[_nMover](
                Axis          := _AxisRefMover[_nMover], 
                Execute       := FALSE, 
                Deceleration  := 15_000, 
                Jerk          := 150_000, 
                BufferMode    := MC_BufferMode.MC_Aborting,
                Error=> , 
                ErrorID=> );
    END_FOR
END_CASE

//-----------------------------------------------------------------------------
//-----------------------------------------------------------------------------

McHaltAll                     := _eState;
END_METHOD

METHOD McResetAll : E_PROGRESS
VAR_INPUT
  Execute       : BOOL;
END_VAR
VAR_INST
  _nErrorId     : UDINT;
  _eState       : E_PROGRESS;

  _nMover       : UINT;
END_VAR
IF NOT Execute THEN _eState     := E_PROGRESS.PROGRESS_INIT; END_IF 
IF NOT Check() THEN McResetAll  := E_PROGRESS.PROGRESS_ERROR; RETURN; END_IF


CASE _eState
OF
  E_PROGRESS.PROGRESS_INIT:
    IF Execute
    THEN
      _nErrorId               := 0;
      _nMover                 := 1;
      _eState                 := E_PROGRESS.PROGRESS_BUSY;
    END_IF
END_CASE
//-----------------------------------------------------------------------------
//-----------------------------------------------------------------------------
CASE _eState
OF
  E_PROGRESS.PROGRESS_BUSY:
    _eState                   := E_PROGRESS.PROGRESS_PREPARE;
    FOR _nMover := 1 TO MAX_MOVER
    DO
      _fbReset[_nMover](
                Axis          := _AxisRefMover[_nMover], 
                Execute       := FALSE);
    END_FOR
END_CASE
//-----------------------------------------------------------------------------
//-----------------------------------------------------------------------------
CASE _eState
OF
  E_PROGRESS.PROGRESS_PREPARE:
    _GroupCommon              := _GroupRef.NcToPlc.Common;
    IF (_GroupCommon.GroupStatus.Flags.AllAxesStanding)
    THEN
      _eState                 := E_PROGRESS.PROGRESS_CHECK;
    END_IF

    FOR _nMover := 1 TO MAX_MOVER
    DO
      _fbReset[_nMover](
                Axis          := _AxisRefMover[_nMover], 
                Execute       := TRUE);

      IF (_fbReset[_nMover].Error)
      THEN
        _nErrorId             := _fbReset[_nMover].ErrorID;
        _eState               := E_PROGRESS.PROGRESS_ERROR;
        EXIT;
      END_IF
    END_FOR
END_CASE
//-----------------------------------------------------------------------------
//-----------------------------------------------------------------------------
CASE _eState
OF
  E_PROGRESS.PROGRESS_CHECK:
    _eState                   := E_PROGRESS.PROGRESS_DONE;
    FOR _nMover := 1 TO MAX_MOVER
    DO
      _fbReset[_nMover](
                Axis          := _AxisRefMover[_nMover], 
                Execute       := FALSE);
    END_FOR
END_CASE
//-----------------------------------------------------------------------------
//-----------------------------------------------------------------------------

McResetAll                    := _eState;
END_METHOD

METHOD RemoveAll : E_PROGRESS
VAR_INPUT
  Execute     : BOOL;
END_VAR
VAR_INST
  _nErrorId   : UDINT;
  _eState     : E_PROGRESS;

  _nMover     : UINT;
END_VAR
IF NOT Execute THEN _eState         := E_PROGRESS.PROGRESS_INIT; END_IF 
IF NOT Check() THEN RemoveAll  := E_PROGRESS.PROGRESS_ERROR; RETURN; END_IF


CASE _eState
OF
  E_PROGRESS.PROGRESS_INIT:
    IF Execute
    THEN
      _nErrorId               := 0;
      _nMover                 := 1;
      _GroupCommon            := _GroupRef.NcToPlc.Common;

      IF (_GroupCommon.GroupAxesCount > 0)
      THEN
        _eState               := E_PROGRESS.PROGRESS_BUSY;
      ELSE
        _eState               := E_PROGRESS.PROGRESS_DONE;
      END_IF
    END_IF
END_CASE
//-----------------------------------------------------------------------------
//-----------------------------------------------------------------------------
CASE _eState
OF
  E_PROGRESS.PROGRESS_BUSY:
    _eState                   := E_PROGRESS.PROGRESS_PREPARE;
    _fbRemoveAxisGroup[_nMover](
              AxesGroup       := _GroupRef, 
              Execute         := FALSE,
              IdentInGroup    := UDINT_TO_IDENTINGROUP(_AxisRefMover[_nMover].NcToPlc.AxisId));
END_CASE
//-----------------------------------------------------------------------------
//-----------------------------------------------------------------------------
CASE _eState
OF
  E_PROGRESS.PROGRESS_PREPARE:
    _fbRemoveAxisGroup[_nMover](
              AxesGroup       := _GroupRef, 
              Execute         := TRUE,
              IdentInGroup    := UDINT_TO_IDENTINGROUP(_AxisRefMover[_nMover].NcToPlc.AxisId));

    IF (_fbRemoveAxisGroup[_nMover].Error)
    THEN
      _eState                 := E_PROGRESS.PROGRESS_ERROR;
      _nErrorId               := _fbRemoveAxisGroup[_nMover].ErrorId;

    ELSIF (_fbRemoveAxisGroup[_nMover].Done)
    THEN
      _eState                 := E_PROGRESS.PROGRESS_CHECK;
    END_IF
END_CASE
//-----------------------------------------------------------------------------
//-----------------------------------------------------------------------------
CASE _eState
OF
  E_PROGRESS.PROGRESS_CHECK:
    _eState                   := E_PROGRESS.PROGRESS_OCCUPIED;
    _fbRemoveAxisGroup[_nMover](
              AxesGroup       := _GroupRef, 
              Execute         := FALSE,
              IdentInGroup    := UDINT_TO_IDENTINGROUP(_AxisRefMover[_nMover].NcToPlc.AxisId));
END_CASE
//-----------------------------------------------------------------------------
//-----------------------------------------------------------------------------
CASE _eState
OF
  E_PROGRESS.PROGRESS_OCCUPIED:
    _nMover                   := _nMover + 1;

    IF NOT (_nMover > MAX_MOVER)
    THEN
      _eState                 := E_PROGRESS.PROGRESS_BUSY;
    ELSE
      _eState                 := E_PROGRESS.PROGRESS_DONE;
    END_IF
END_CASE
//-----------------------------------------------------------------------------
//-----------------------------------------------------------------------------

RemoveAll                := _eState;
END_METHOD

METHOD Reset : E_PROGRESS
VAR_INPUT
  Execute     : BOOL;
END_VAR
VAR_INST
  _nErrorId   : UDINT;
  _eState     : E_PROGRESS;

  _nMover     : UINT;
END_VAR
IF NOT Execute 
THEN 
	_eState := E_PROGRESS.PROGRESS_INIT; 
END_IF 
IF NOT Check() 
THEN 
	Reset := E_PROGRESS.PROGRESS_ERROR; 
	RETURN; 
END_IF


CASE _eState
OF
  E_PROGRESS.PROGRESS_INIT:
    IF Execute
    THEN
      _nErrorId                 := 0;
      _nMover                   := 1;
      _stGroupInfo.GroupErrorId := 0;
      _stGroupInfo.GroupError   := FALSE;

      _eState                   := E_PROGRESS.PROGRESS_BUSY;
    END_IF
END_CASE
//-----------------------------------------------------------------------------
//-----------------------------------------------------------------------------
CASE _eState
OF
  E_PROGRESS.PROGRESS_BUSY:
    _eState                     := E_PROGRESS.PROGRESS_PREPARE;
    _fbGroupReset(
              AxesGroup         := _GroupRef, 
              Execute           := FALSE);
END_CASE
//-----------------------------------------------------------------------------
//-----------------------------------------------------------------------------
CASE _eState
OF
  E_PROGRESS.PROGRESS_PREPARE:
    _fbGroupReset(
              AxesGroup         := _GroupRef, 
              Execute           := TRUE);

    IF (_fbGroupReset.Error)
    THEN
      _eState                   := E_PROGRESS.PROGRESS_ERROR;
      _nErrorId                 := _fbGroupReset.ErrorId;
      _fbGroupReset(
              AxesGroup         := _GroupRef, 
              Execute           := FALSE); 


    ELSIF (_fbGroupReset.Done)
    THEN
      _eState                   := E_PROGRESS.PROGRESS_DONE;
      _fbGroupReset(
              AxesGroup         := _GroupRef, 
              Execute           := FALSE); 
    END_IF
END_CASE
//-----------------------------------------------------------------------------
//-----------------------------------------------------------------------------

Reset                           := _eState;
END_METHOD

END_FUNCTION_BLOCK

// ---- XTS/CaGroup/old/fb_GroupCtrl.TcPOU
//---------------------------------------------------------------------------------------------------------------
//
//  HAUD 2023.12.13
//
//
//  fb_GroupCtrl
//  - procedures for getting group ready to work
//
//
//  CTRL / STATE --> see proprerties
//  structs for use of function block via mapping
//  cyclic check for new command
//
//  VAR INPUT / OUTPUT --> see properties
//
//---------------------------------------------------------------------------------------------------------------
// This SOFTWARE is provided as an Exemple by THE PROVIDER "as is" and "with all faults." THE PROVIDER makes no 
// representations or warranties of any kind concerning the safety, suitability, lack of viruses, inaccuracies, 
// typographical errors, or other harmful components of this SOFTWARE. There are inherent dangers in the use of 
// any software, and you are solely responsible for determining whether this SOFTWARE is compatible with your 
// equipment and other software installed on your equipment. You are also solely responsible for the protection 
// of your equipment and backup of your data, and THE PROVIDER will not be liable for any damages you may suffer 
// in connection with using, modifying, or distributing this SOFTWARE.
//---------------------------------------------------------------------------------------------------------------
FUNCTION_BLOCK fb_GroupCtrl EXTENDS FB_CaGroup
VAR
  _stCtrl                     : REFERENCE TO ST_GROUP_CTRL;
  _stState                    : REFERENCE TO ST_GROUP_STATE;

  _eCmd,
  _eCmdOld                    : E_GROUP_CTRL;

  _eResult                    : E_PROGRESS;
  _eState                     : E_GROUP_STATE;

  _wGroupState                : DWORD;
END_VAR

IF NOT Check() THEN RETURN; END_IF

// copy to local for ease of use with breadcrums
_GroupCommon                  := _GroupRef.NcToPlc.Common;


// copy to local for debug
_eCmd                         := _stCtrl.Cmd;

// cyclic check for command change
// get state for cmd
IF (_eCmd <> _eCmdOld)
THEN
  // get matching sdtate for Ctrl.Cmd
  _eState                     := Cmd(_eCmd);
  _eCmdOld                    := _eCmd;
END_IF


CASE _eState
OF
  E_GROUP_STATE.GROUP_CLEAR:
    // halt all mover
    // remove all mover from group
    // reset all mover
    // disable group
    // reset group
    _eResult                  := GroupClear(TRUE);

  E_GROUP_STATE.GROUP_BUILD:
    // halt all mover
    // reset all mover
    // check for empty group (must be empty, since we want to build it now)
    // reset group
    // add all mover to group
    _eResult                  := GroupBuild(TRUE);

  E_GROUP_STATE.GROUP_ENABLE:
    // reset all mover
    // reset group
    // check if group has movers (group must have been built before)
    // enable group
    // wait for mcGroupStateStandby or mcGroupStateMoving
    _eResult                  := GroupEnable(TRUE);

ELSE
  _eResult                    := E_GROUP_STATE.GROUP_INVALID;
END_CASE

_stState.McState            := _GroupCommon.GroupStatus;
_stState.AxisCount          := TO_UINT(_GroupCommon.GroupAxesCount);

// cyclic MC_GroupReadStatus check
// cyclic MC_GroupReadError check
_wGroupState                := InfoCycle(TRUE);
IF NOT _wGroupState.13 
THEN
  // in case of error, tell everyone
  _eResult                  := E_PROGRESS.PROGRESS_ERROR;
END_IF


CASE _eResult
OF
  E_PROGRESS.PROGRESS_INVALID:
    _stState.State            := _eResult;

  E_PROGRESS.PROGRESS_ERROR:
    _stState.State            := _eState + E_PROGRESS.PROGRESS_ERROR;

  E_PROGRESS.PROGRESS_DONE:
    _stState.State            := _eState + E_PROGRESS.PROGRESS_DONE;

ELSE
  // work in progress
  // update progress for extern use
  _stState.State              := _eState + _eResult;
END_CASE

METHOD Check : BOOL

IF NOT __ISVALIDREF(_GroupRef)
THEN
  _eCheck                     := E_GROUP_CHECK.CHECK_GROUP_REF_INVALID;
  RETURN;
END_IF

IF NOT __ISVALIDREF(_AxisRefMover)
THEN
  _eCheck                     := E_GROUP_CHECK.CHECK_AXIS_REF_INVALID;
  RETURN;
END_IF

IF NOT __ISVALIDREF(_stCtrl)
THEN
  _eCheck                     := E_GROUP_CHECK.CHECK_CTRL_INVALID;
  RETURN;
END_IF

IF NOT __ISVALIDREF(_stState)
THEN
  _eCheck                     := E_GROUP_CHECK.CHECK_STATE_INVALID;
  RETURN;
END_IF


_eCheck                       := E_GROUP_CHECK.CHECK_DONE;
Check                         := TRUE;
END_METHOD

METHOD PRIVATE Cmd : E_GROUP_STATE
VAR_INPUT
  Ctrl      : E_GROUP_CTRL;
END_VAR
VAR_INST
  _eState   : E_GROUP_STATE;
END_VAR
IF NOT Check() THEN RETURN; END_IF


CASE Ctrl
OF
  E_GROUP_CTRL.GROUP_CLEAR:
    GroupClear(FALSE);
    _eState         := E_GROUP_STATE.GROUP_CLEAR;

  E_GROUP_CTRL.GROUP_BUILD:
    GroupBuild(FALSE);
    _eState         := E_GROUP_STATE.GROUP_BUILD;

  E_GROUP_CTRL.GROUP_ENABLE:
    GroupEnable(FALSE);
    _eState         := E_GROUP_STATE.GROUP_ENABLE;

ELSE
    _eState         := E_GROUP_STATE.GROUP_INVALID;
END_CASE

Cmd                 := _eState;
END_METHOD

PROPERTY Ctrl : REFERENCE TO st_group_ctrl
SET
_stCtrl := Ctrl;
END_SET
END_PROPERTY

METHOD GroupBuild : E_PROGRESS
VAR_INPUT
  Execute         : BOOL;
END_VAR
VAR_INST
  _nErrorId   : UDINT;

  _eResult,
  _eState     : E_PROGRESS;

  _nMover     : UINT;
END_VAR
IF NOT Execute THEN _eState     := E_PROGRESS.PROGRESS_INIT; END_IF
IF NOT Check() THEN GroupBuild  := E_PROGRESS.PROGRESS_ERROR; RETURN; END_IF


CASE _eState
OF
  E_PROGRESS.PROGRESS_INIT:
    IF Execute
    THEN
      _nErrorId               := 0;
      _eState                 := E_PROGRESS.PROGRESS_BUSY;
      _eResult                := McHaltAll(FALSE);
    END_IF
END_CASE
//-----------------------------------------------------------------------------
//-----------------------------------------------------------------------------
CASE _eState
OF
  E_PROGRESS.PROGRESS_BUSY:
    _eResult                  := McHaltAll(TRUE);

    IF (_eResult = E_PROGRESS.PROGRESS_ERROR)
    THEN
      _eState                 := E_PROGRESS.PROGRESS_ERROR;
      _eResult                := McHaltAll(FALSE);

    ELSIF (_eResult = E_PROGRESS.PROGRESS_DONE)
    THEN
      _eState                 := E_PROGRESS.PROGRESS_PREPARE;
      _eResult                := McHaltAll(FALSE);
      _eResult                := McResetAll(FALSE);
    END_IF
END_CASE
//-----------------------------------------------------------------------------
//-----------------------------------------------------------------------------
CASE _eState
OF
  E_PROGRESS.PROGRESS_PREPARE:
    _eResult                  := McResetAll(TRUE);

    IF (_eResult = E_PROGRESS.PROGRESS_ERROR)
    THEN
      _eState                 := E_PROGRESS.PROGRESS_ERROR;
      _eResult                := McResetAll(FALSE);

    ELSIF (_eResult = E_PROGRESS.PROGRESS_DONE)
    THEN
      _eState                 := E_PROGRESS.PROGRESS_STARTUP;
      _eResult                := McResetAll(FALSE);
    END_IF
END_CASE
//-----------------------------------------------------------------------------
//-----------------------------------------------------------------------------
CASE _eState
OF
  E_PROGRESS.PROGRESS_STARTUP:
    IF (_GroupCommon.GroupAxesCount <> 0)
    THEN
      _nErrorId               := _eState;
      _eState                 := E_PROGRESS.PROGRESS_ERROR;
    ELSE
      _eState                 := E_PROGRESS.PROGRESS_CHECK;
      _eResult                := Reset(FALSE);
    END_IF
END_CASE
//-----------------------------------------------------------------------------
//-----------------------------------------------------------------------------
CASE _eState
OF
  E_PROGRESS.PROGRESS_CHECK:
    _eResult                  := Reset(TRUE);

    IF (_eResult = E_PROGRESS.PROGRESS_ERROR)
    THEN
      _eState                 := E_PROGRESS.PROGRESS_ERROR;
      _eResult                := Reset(FALSE);

    ELSIF (_eResult = E_PROGRESS.PROGRESS_DONE)
    THEN
      _eState                 := E_PROGRESS.PROGRESS_OCCUPIED;
      _eResult                := Reset(FALSE);
      _eResult                := AddAll(FALSE);
    END_IF
END_CASE
//-----------------------------------------------------------------------------
//-----------------------------------------------------------------------------
CASE _eState
OF
  E_PROGRESS.PROGRESS_OCCUPIED:
    _eResult                  := AddAll(TRUE);

    IF (_eResult = E_PROGRESS.PROGRESS_ERROR)
    THEN
      _eState                 := E_PROGRESS.PROGRESS_ERROR;
      _eResult                := AddAll(FALSE);

    ELSIF (_eResult = E_PROGRESS.PROGRESS_DONE)
    THEN
      _eState                 := E_PROGRESS.PROGRESS_WORKING;
      _eResult                := AddAll(FALSE);
    END_IF
END_CASE
//-----------------------------------------------------------------------------
//-----------------------------------------------------------------------------
CASE _eState
OF
  E_PROGRESS.PROGRESS_WORKING:
    IF (_GroupCommon.GroupStatus.State = mcGroupStateDisabled)
    THEN
      _eState                 := E_PROGRESS.PROGRESS_DONE;
    END_IF
END_CASE
//-----------------------------------------------------------------------------
//-----------------------------------------------------------------------------

GroupBuild                    := _eState;
END_METHOD

METHOD GroupClear : E_PROGRESS
VAR_INPUT
  Execute         : BOOL;
END_VAR
VAR_INST
  _nErrorId   : UDINT;

  _eResult,
  _eState     : E_PROGRESS;

  _nMover     : UINT;
END_VAR
IF NOT Execute THEN _eState     := E_PROGRESS.PROGRESS_INIT; END_IF
IF NOT Check() THEN GroupClear  := E_PROGRESS.PROGRESS_ERROR; RETURN; END_IF


CASE _eState
OF
  E_PROGRESS.PROGRESS_INIT:
    IF Execute
    THEN
      _nErrorId               := 0;
      _eState                 := E_PROGRESS.PROGRESS_BUSY;
      _eResult                := McHaltAll(FALSE);
    END_IF
END_CASE
//-----------------------------------------------------------------------------
//-----------------------------------------------------------------------------
CASE _eState
OF
  E_PROGRESS.PROGRESS_BUSY:
    _eResult                  := McHaltAll(TRUE);

    IF (_eResult = E_PROGRESS.PROGRESS_ERROR)
    THEN
      _eState                 := E_PROGRESS.PROGRESS_ERROR;
      _eResult                := McHaltAll(FALSE);

    ELSIF (_eResult = E_PROGRESS.PROGRESS_DONE)
    THEN
      _eState                 := E_PROGRESS.PROGRESS_PREPARE;
      _eResult                := McHaltAll(FALSE);
    END_IF
END_CASE
//-----------------------------------------------------------------------------
//-----------------------------------------------------------------------------
CASE _eState
OF
  E_PROGRESS.PROGRESS_PREPARE:
    IF (_GroupCommon.GroupStatus.State = mcGroupStateErrorStop)
    THEN
      _eState                 := E_PROGRESS.PROGRESS_STARTUP;
      _eResult                := McResetAll(FALSE);

    ELSE
      _eState                 := E_PROGRESS.PROGRESS_CHECK;
      _eResult                := RemoveAll(FALSE);
    END_IF
END_CASE
//-----------------------------------------------------------------------------
//-----------------------------------------------------------------------------
CASE _eState
OF
  E_PROGRESS.PROGRESS_STARTUP:
    _eResult                  := McResetAll(TRUE);

    IF (_eResult = E_PROGRESS.PROGRESS_ERROR)
    THEN
      _eState                 := E_PROGRESS.PROGRESS_ERROR;
      _eResult                := McResetAll(FALSE);

    ELSIF (_eResult = E_PROGRESS.PROGRESS_DONE)
    THEN
      _eState                 := E_PROGRESS.PROGRESS_CHECK;
      _eResult                := McResetAll(FALSE);
      _eResult                := RemoveAll(FALSE);
    END_IF
END_CASE
//-----------------------------------------------------------------------------
//-----------------------------------------------------------------------------
CASE _eState
OF
  E_PROGRESS.PROGRESS_CHECK:
    _eResult                  := RemoveAll(TRUE);

    IF (_eResult = E_PROGRESS.PROGRESS_ERROR)
    THEN
      _eState                 := E_PROGRESS.PROGRESS_ERROR;
      _eResult                := RemoveAll(FALSE);

    ELSIF (_eResult = E_PROGRESS.PROGRESS_DONE)
    THEN
      _eState                 := E_PROGRESS.PROGRESS_OCCUPIED;
      _eResult                := RemoveAll(FALSE);
      _eResult                := Disable(FALSE);
    END_IF
END_CASE
//-----------------------------------------------------------------------------
//-----------------------------------------------------------------------------
CASE _eState
OF
  E_PROGRESS.PROGRESS_OCCUPIED:
    _eResult                  := Disable(TRUE);

    IF (_eResult = E_PROGRESS.PROGRESS_ERROR)
    THEN
      _eState                 := E_PROGRESS.PROGRESS_ERROR;
      _eResult                := Disable(FALSE);

    ELSIF (_eResult = E_PROGRESS.PROGRESS_DONE)
    THEN
      _eState                 := E_PROGRESS.PROGRESS_WORKING;
      _eResult                := Disable(FALSE);
      _eResult                := Reset(FALSE);
    END_IF
END_CASE
//-----------------------------------------------------------------------------
//-----------------------------------------------------------------------------
CASE _eState
OF
  E_PROGRESS.PROGRESS_WORKING:
    _eResult                  := Reset(TRUE);

    IF (_eResult = E_PROGRESS.PROGRESS_ERROR)
    THEN
      _eState                 := E_PROGRESS.PROGRESS_ERROR;
      _eResult                := Reset(FALSE);

    ELSIF (_eResult = E_PROGRESS.PROGRESS_DONE)
    THEN
      _eState                 := E_PROGRESS.PROGRESS_DONE;
      _eResult                := Reset(FALSE);
    END_IF
END_CASE
//-----------------------------------------------------------------------------
//-----------------------------------------------------------------------------

GroupClear                    := _eState;
END_METHOD

METHOD PRIVATE GroupEnable : E_PROGRESS
VAR_INPUT
  Execute         : BOOL;
END_VAR
VAR_INST
  _nErrorId   : UDINT;

  _eResult,
  _eState     : E_PROGRESS;

  _nMover     : UINT;
END_VAR
IF NOT Execute THEN _eState     := E_PROGRESS.PROGRESS_INIT; END_IF
IF NOT Check() THEN GroupEnable := E_PROGRESS.PROGRESS_ERROR; RETURN; END_IF


CASE _eState
OF
  E_PROGRESS.PROGRESS_INIT:
    IF Execute
    THEN
      _nErrorId               := 0;
      _eState                 := E_PROGRESS.PROGRESS_BUSY;
      _eResult                := McResetAll(FALSE);
    END_IF
END_CASE
//-----------------------------------------------------------------------------
//-----------------------------------------------------------------------------
CASE _eState
OF
  E_PROGRESS.PROGRESS_BUSY:
    _eResult                  := McResetAll(TRUE);

    IF (_eResult = E_PROGRESS.PROGRESS_ERROR)
    THEN
      _eState                 := E_PROGRESS.PROGRESS_ERROR;
      _eResult                := McResetAll(FALSE);

    ELSIF (_eResult = E_PROGRESS.PROGRESS_DONE)
    THEN
      _eState                 := E_PROGRESS.PROGRESS_PREPARE;
      _eResult                := McResetAll(FALSE);
    END_IF
END_CASE
//-----------------------------------------------------------------------------
//-----------------------------------------------------------------------------
CASE _eState
OF
  E_PROGRESS.PROGRESS_PREPARE:
    _eResult                  := Reset(TRUE);

    IF (_eResult = E_PROGRESS.PROGRESS_ERROR)
    THEN
      _eState                 := E_PROGRESS.PROGRESS_ERROR;
      _eResult                := Reset(FALSE);

    ELSIF (_eResult = E_PROGRESS.PROGRESS_DONE)
    THEN
      _eState                 := E_PROGRESS.PROGRESS_OCCUPIED;
      _eResult                := Reset(FALSE);
    END_IF
END_CASE
//-----------------------------------------------------------------------------
//-----------------------------------------------------------------------------
CASE _eState
OF
  E_PROGRESS.PROGRESS_STARTUP:
    IF NOT (_GroupCommon.GroupAxesCount <> 0)
    THEN
      _nErrorId               := _eState;
      _eState                 := E_PROGRESS.PROGRESS_ERROR;
    ELSE
      _eState                 := E_PROGRESS.PROGRESS_CHECK;
      _eResult                := Enable(FALSE);
    END_IF
END_CASE
//-----------------------------------------------------------------------------
//-----------------------------------------------------------------------------
CASE _eState
OF
  E_PROGRESS.PROGRESS_CHECK:
    _eResult                  := Enable(TRUE);

    IF (_eResult = E_PROGRESS.PROGRESS_ERROR)
    THEN
      _eState                 := E_PROGRESS.PROGRESS_ERROR;
      _eResult                := Enable(FALSE);

    ELSIF (_eResult = E_PROGRESS.PROGRESS_DONE)
    THEN
      _eState                 := E_PROGRESS.PROGRESS_WORKING;
      _eResult                := Enable(FALSE);
    END_IF
END_CASE
//-----------------------------------------------------------------------------
//-----------------------------------------------------------------------------
CASE _eState
OF
  E_PROGRESS.PROGRESS_WORKING:
    IF (_GroupCommon.GroupStatus.State = mcGroupStateStandby) OR
       (_GroupCommon.GroupStatus.State = mcGroupStateMoving)
    THEN
      _eState                 := E_PROGRESS.PROGRESS_DONE;
    END_IF
END_CASE
//-----------------------------------------------------------------------------
//-----------------------------------------------------------------------------

GroupBuild                    := _eState;
END_METHOD

PROPERTY State : REFERENCE TO ST_GROUP_STATE
SET
_stState := State;
END_SET
END_PROPERTY

END_FUNCTION_BLOCK

// ---- VISUs/CA_Visu.TcVIS
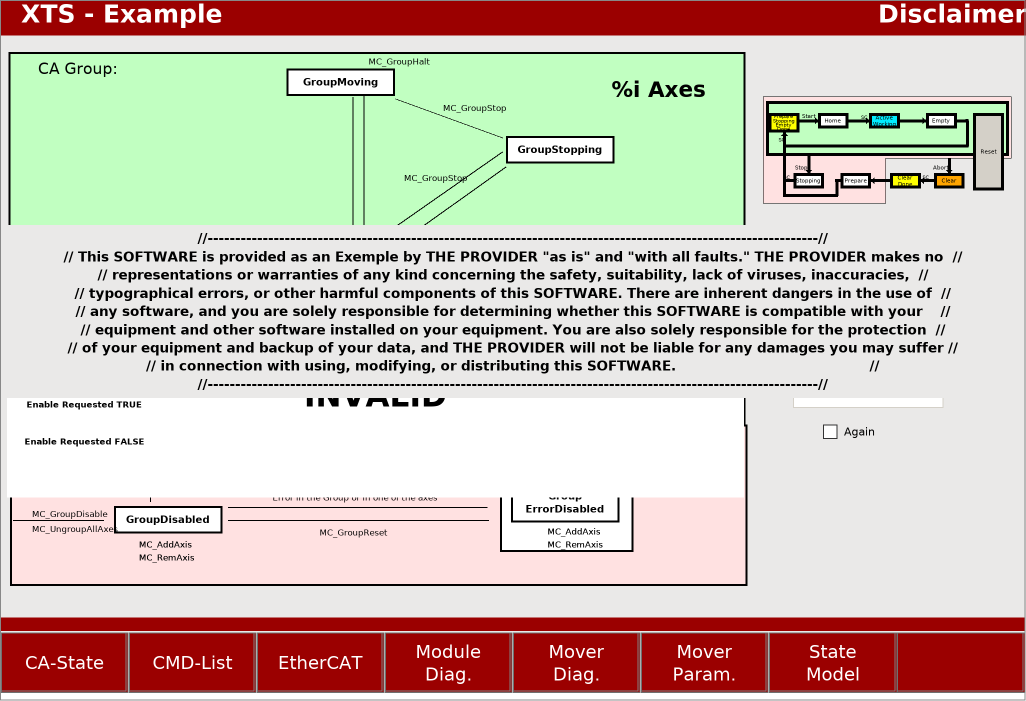
VISUALIZATION CA_Visu  // 1026x701
VAR_IN_OUT
	
END_VAR

VAR
	bShowDisclaimer		: BOOL;
END_VAR
    Frame (0,-8 1026x701)
        shows FrameVisuSimpelCaExample(stVisuIO := MAIN.fbSimpleCaMove.stVisuIO)
END_VISUALIZATION

// ---- VISUs/Frame/FrameVisuSimpelCaExample.TcVIS
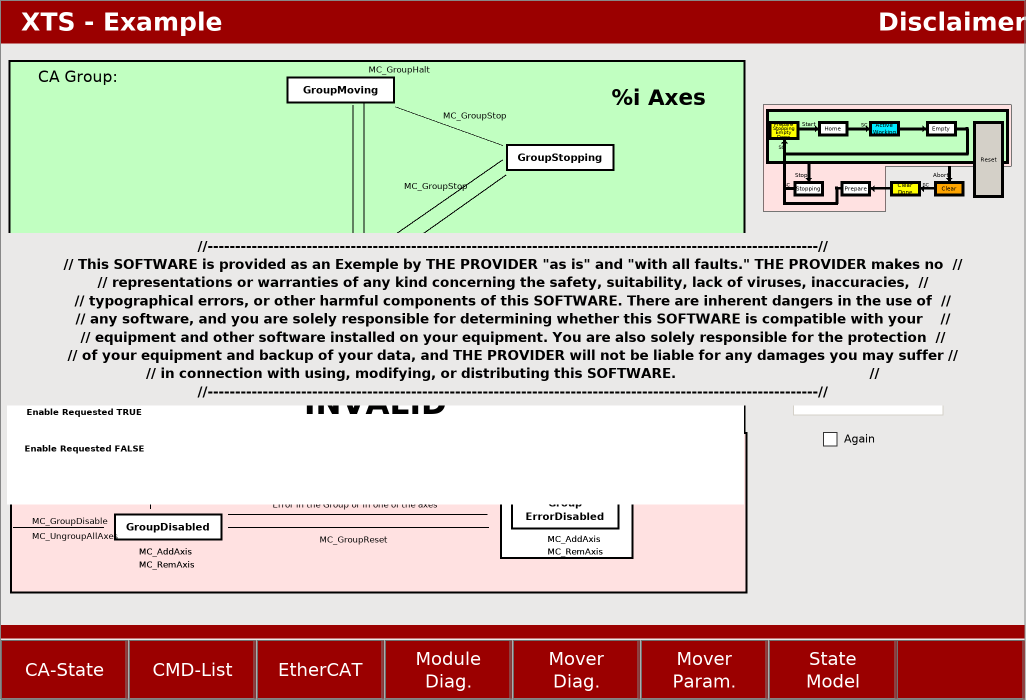
VISUALIZATION FrameVisuSimpelCaExample  // 1026x700
VAR_IN_OUT
	
	stVisuIO		: ST_VisuExampleIO;


	
END_VAR

VAR
	sVisuXtsDiag		: STRING := 'Visu_XtsDiag';
	nFrameSelect		: INT;
	
	bShowDisclaimer		: BOOL;
END_VAR
    Rectangle (1,0 1024x43), "XTS - Example"
    Rectangle (1,625 1024x13)
    Button (1,640 127x60), "CA-State", input disabled if: nFrameSelect = 0
        OnMouseClick: execute { nFrameSelect := 0; }
    Button (129,640 127x60), "CMD-List", input disabled if: (nFrameSelect = 1) or true
        OnMouseClick: execute { nFrameSelect := 1; }
    Button (257,640 127x60), "EtherCAT", input disabled if: (nFrameSelect =2) or true
        OnMouseClick: execute { nFrameSelect := 2; }
    Button (385,640 127x60), "Module Diag.", input disabled if: (nFrameSelect = 3) or true
        OnMouseClick: execute { nFrameSelect := 3; }
    Button (513,640 127x60), "Mover Diag.", input disabled if: (nFrameSelect = 4) or true
        OnMouseClick: execute { nFrameSelect := 4; }
    Button (641,640 127x60), "Mover Param.", input disabled if: (nFrameSelect = 5) or true
        OnMouseClick: execute { nFrameSelect := 5; }
    Button (897,640 128x60)
    Button (769,640 128x60), "State Model", input disabled if: nFrameSelect = 6
        OnMouseClick: execute { nFrameSelect:= 6; }
    Textfield (793,312 150x30), "Set Pos1: %.2f", text variable: stVisuIO.fSetPos1
        OnMouseClick: write the text variable via Default, min 0, max 50000
    Textfield (793,348 150x30), "Set Pos2: %.2f", text variable: stVisuIO.fSetPos2
        OnMouseClick: write the text variable via Default, min 0, max 50000
    Checkbox (821,424 94x30), "Again", variable: stVisuIO.bAgain
    Textfield (793,385 150x30), "Set Pos3: %.2f", text variable: stVisuIO.fSetPos3
        OnMouseClick: write the text variable via Default, min 0, max 50000
    Frame (7,60 740x533), frame switch variable: nFrameSelect
        shows FrameAdvancedMotion(stCaGroup := stVisuIO.stCaGroup)
        shows FrameDummy()
        shows FrameDummy()
        shows FrameDummy()
        shows FrameDummy()
        shows FrameDummy()
        shows FrameXtsStateModel(eOPMState := stVisuIO.eOPMState, eStateCommand := stVisuIO.eStateCommand)
    Frame (757,71 260x174), frame switch variable: nFrameSelect
        shows FrameXtsStateModel(eOPMState := stVisuIO.eOPMState, eStateCommand := stVisuIO.eStateCommand)
        shows FrameXtsStateModel(eOPMState := stVisuIO.eOPMState, eStateCommand := stVisuIO.eStateCommand)
        shows FrameXtsStateModel(eOPMState := stVisuIO.eOPMState, eStateCommand := stVisuIO.eStateCommand)
        shows FrameXtsStateModel(eOPMState := stVisuIO.eOPMState, eStateCommand := stVisuIO.eStateCommand)
        shows FrameXtsStateModel(eOPMState := stVisuIO.eOPMState, eStateCommand := stVisuIO.eStateCommand)
        shows FrameXtsStateModel(eOPMState := stVisuIO.eOPMState, eStateCommand := stVisuIO.eStateCommand)
        shows FrameAdvancedMotion(stCaGroup := stVisuIO.stCaGroup)
    Rectangle (875,0 151x43), "Disclaimer"
        toggle bShowDisclaimer
    Frame (5,233 1016x172), invisible if: not bShowDisclaimer
        shows FrameDislaimer()
END_VISUALIZATION

// ---- VISUs/Frame/SubFrame/FrameAdvancedMotion.TcVIS
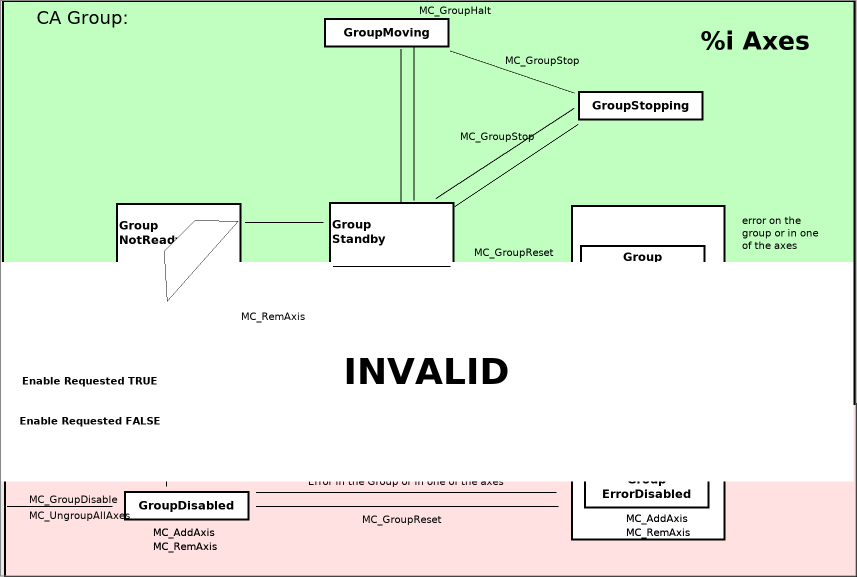
VISUALIZATION FrameAdvancedMotion  // 857x577
VAR_IN_OUT
	stCaGroup			: AXES_GROUP_REF;
END_VAR
    RoundedRectangle (4,403 853x174)
    RoundedRectangle (2,0 853x403)
    RoundedRectangle (324,18 125x29), "GroupMoving", colour toggle: stCaGroup.NcToPlc.Common.GroupStatus.State = 3
    RoundedRectangle (329,202 125x100), "Group Standby", colour toggle: stCaGroup.NcToPlc.Common.GroupStatus.State = 2
    RoundedRectangle (578,91 125x29), "GroupStopping", colour toggle: stCaGroup.NcToPlc.Common.GroupStatus.State = 4
    RoundedRectangle (116,203 125x100), "Group NotReady", colour toggle: stCaGroup.NcToPlc.Common.GroupStatus.State = 7
    RoundedRectangle (571,205 154x335), "GroupErrorStop", colour toggle: stCaGroup.NcToPlc.Common.GroupStatus.State = 5
    RoundedRectangle (124,491 125x29), "GroupDisabled", text variable: stCaGroup.NcToPlc.Common.GroupStatus.State = 1, colour toggle: stCaGroup.NcToPlc.Common.GroupStatus.State = 1
    RoundedRectangle (580,245 125x39), "Group ErrorEnabled"
    RoundedRectangle (584,466 125x42), "Group ErrorDisabled"
    Line (256,506) (558,506)
    Line (167,303) (166,486)
    Line (457,266) (579,266)
    Line (436,198) (574,108)
    Line (414,200) (414,47)
    Group (364,306 62x29)
        Label (0,0 73x15), "MC_AddAxis"
        Label (0,14 74x15), "MC_RemAxis"
    Label (364,306 61x15), "MC_AddAxis"
    Label (364,320 62x15), "MC_RemAxis"
    Group (150,525 62x29)
        Label (0,0 73x15), "MC_AddAxis"
        Label (0,14 74x15), "MC_RemAxis"
    Label (150,525 61x15), "MC_AddAxis"
    Label (150,539 62x15), "MC_RemAxis"
    Group (172,308 62x29)
        Label (0,0 73x15), "MC_AddAxis"
        Label (0,14 74x15), "MC_RemAxis"
    Label (172,308 61x15), "MC_AddAxis"
    Label (172,322 62x15), "MC_RemAxis"
    Group (623,511 62x29)
        Label (0,0 73x15), "MC_AddAxis"
        Label (0,14 74x15), "MC_RemAxis"
    Label (623,511 61x15), "MC_AddAxis"
    Label (623,525 62x15), "MC_RemAxis"
    Group (616,286 62x29)
        Label (0,0 73x15), "MC_AddAxis"
        Label (0,14 74x15), "MC_RemAxis"
    Label (616,286 61x15), "MC_AddAxis"
    Label (616,301 62x15), "MC_RemAxis"
    Label (359,512 77x15), "MC_GroupReset"
    Label (471,245 77x15), "MC_GroupReset"
    Label (26,492 77x15), "MC_GroupDisable"
    Label (416,3 77x15), "MC_GroupHalt"
    Label (502,53 77x15), "MC_GroupStop"
    Label (128,431 77x15), "MC_GroupEnable"
    Line (7,506) (112,506)
    Label (26,508 88x15), "MC_UngroupAllAxes"
    Label (247,272 77x22), "one axis not ready"
    Label (739,215 77x36), "error on the group or in one of the axes"
    Line (401,202) (401,49)
    Line (455,206) (578,124)
    Line (256,492) (556,492)
    Line (245,222) (323,222)
    Label (305,474 170x15), "Error in the Group or in one of the axes"
    Line (233,480) (342,309), "MC_GroupStop"
    Line (234,478) (236,306), "MC_GroupStop"
    Line (246,266) (324,266)
    Line (574,93) (450,51)
    Group (590,294 11x164)
        Line (6,150) (6,0)
        Line (6,161) (13,146)
        Line (5,161) (0,146)
    Line (595,445) (595,293)
    Line (595,457) (600,441)
    Line (594,457) (590,441)
    Group (693,295 11x164)
        Line (6,150) (6,0)
        Line (6,161) (13,146)
        Line (5,161) (0,146)
    Line (698,446) (698,294)
    Line (698,458) (704,442)
    Line (697,458) (693,442)
    Rectangle (0,262 853x219), "INVALID", invisible if: stCaGroup.NcToPlc.Common.GroupStatus.State <> 0
    Label (14,366 152x30), "Enable Requested TRUE", invisible if: stCaGroup.NcToPlc.Common.GroupStatus.Flags.IsEnableRequested = FALSE
    Label (14,406 152x30), "Enable Requested FALSE", invisible if: stCaGroup.NcToPlc.Common.GroupStatus.Flags.IsEnableRequested = TRUE
    Label (457,129 77x15), "MC_GroupStop"
    Polygon (167,301) (164,251) (195,220) (227,221) (238,221)
    Line (333,266) (450,266)
    Label (238,309 60x15), "MC_RemAxis"
    Rectangle (695,10 118x61), "%i Axes", text variable: stCaGroup.NcToPlc.CA.Common.GroupAxesCount
    Rectangle (34,6 97x24), "CA Group:"
END_VISUALIZATION

// ---- VISUs/Frame/SubFrame/FrameDummy.TcVIS
VISUALIZATION FrameDummy  // 2x2
END_VISUALIZATION

// ---- VISUs/Frame/SubFrame/FrameXtsStateModel.TcVIS
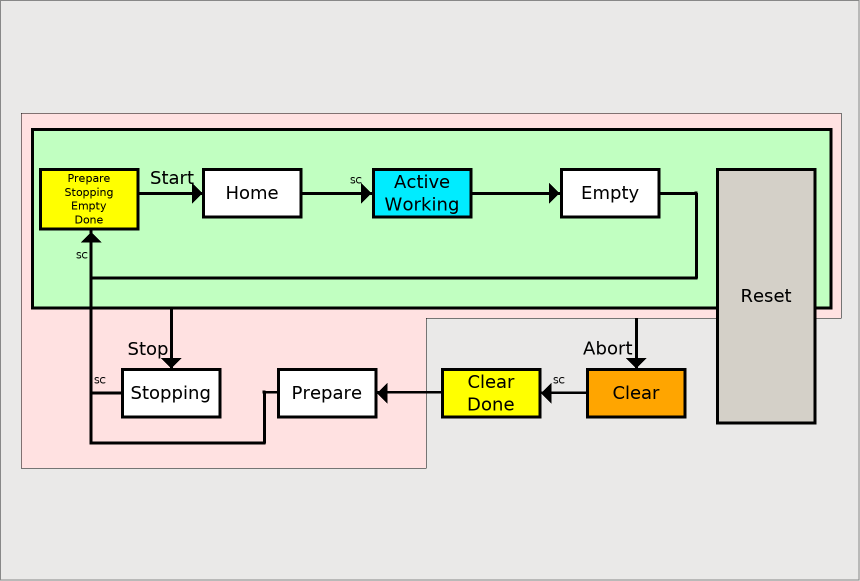
VISUALIZATION FrameXtsStateModel  // 860x581
VAR_IN_OUT

	eOPMState			: E_OperatingState;
	eStateCommand		: E_OperatingCmd;
	
END_VAR
    Rectangle (-10,1 860x580)
    Polygon (21,113) (841,113) (841,318) (426,318) (426,468) (21,468)
    Rectangle (31,128 801x181)
    Polyline (636,318) (636,393) (264,392) (264,443) (191,443) (91,443) (91,393) (91,193) (411,193)
    RoundedRectangle (39,168 100x62), "Prepare Stopping Empty Done", colour toggle: eOPMState = E_OperatingState.OperatingMode_Prepar_Sc
    RoundedRectangle (202,168 100x50), "Home", colour toggle: (eOPMState = E_OperatingState.OperatingMode_Home)
        OnMouseClick: execute { eStateCommand := E_OperatingCmd.OperatingCmd_Home; }
    RoundedRectangle (277,368 100x50), "Prepare", colour toggle: (eOPMState = E_OperatingState.OperatingMode_Prepare)
        OnMouseClick: execute { eStateCommand := E_OperatingCmd.OperatingCmd_Prepare; }
    RoundedRectangle (441,368 100x50), "Clear Done", colour toggle: (eOPMState = E_OperatingState.OperatingMode_Clear_Sc)
    RoundedRectangle (586,368 100x50), "Clear", colour toggle: (eOPMState = E_OperatingState.OperatingMode_Clear)
        OnMouseClick: execute { eStateCommand := E_OperatingCmd.OperatingCmd_Clear; }
    Polygon (91,232) (81,242) (101,242)
    Polygon (541,393) (551,403) (551,383)
    Polygon (377,393) (387,403) (387,383)
    Polygon (202,193) (192,203) (192,183)
    Polygon (371,193) (361,203) (361,183)
    Polygon (559,193) (549,203) (549,183)
    Polygon (646,358) (636,368) (626,358)
    Polygon (181,358) (171,368) (161,358)
    Polyline (171,308) (171,393) (91,393)
    RoundedRectangle (121,368 100x50), "Stopping", colour toggle: (eOPMState = E_OperatingState.OperatingMode_Stopping)
        OnMouseClick: execute { eStateCommand := E_OperatingCmd.OperatingCmd_Stopping; }
    Label (316,173 80x15), "SC"
    Polyline (396,193) (696,193) (696,278) (92,278)
    Label (519,373 80x15), "SC"
    Label (60,373 80x15), "SC"
    Label (108,339 80x20), "Stop"
    Label (568,339 80x19), "Abort"
    Label (42,248 80x15), "SC"
    Label (132,169 80x18), "Start", invisible if: eOPMState <> E_OperatingState.OperatingMode_Prepar_Sc
    RoundedRectangle (560,168 100x50), "Empty", colour toggle: (eOPMState = E_OperatingState.OperatingMode_Empty)
        OnMouseClick: execute { eStateCommand := E_OperatingCmd.OperatingCmd_Empty; }
    RoundedRectangle (716,168 100x256), "Reset", colour toggle: (eOPMState = E_OperatingState.OperatingMode_Reset)
        OnMouseClick: execute { eStateCommand := E_OperatingCmd.OperatingCmd_Reset; }
    RoundedRectangle (372,168 100x50), "Active Working", colour toggle: (eOPMState = E_OperatingState.OperatingMode_Active)
END_VISUALIZATION

// ---- VISUs/Frame/SubFrame/FrameDislaimer.TcVIS
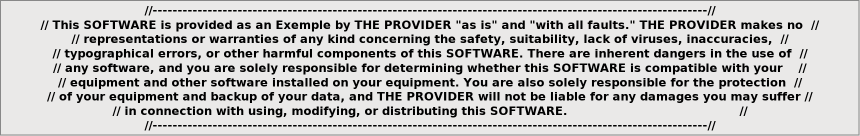
VISUALIZATION FrameDislaimer  // 860x136
    Rectangle (0,0 860x136), "//---------------------------------------------------------------------------------------------------------------// // This SOFTWARE is provided as an Exemple by THE PROVIDER "as is" and "with all faults." THE PROVIDER makes no // // representations or warranties of any kind concerning the safety, suitability, lack of viruses, inaccuracies, // // typographical errors, or other harmful components of this SOFTWARE. There are inherent dangers in the use of // // any software, and you are solely responsible for determining whether this SOFTWARE is compatible with your // // equipment and other software installed on your equipment. You are also solely responsible for the protection // // of your equipment and backup of your data, and THE PROVIDER will not be liable for any damages you may suffer // // in connection with using, modifying, or distributing this SOFTWARE. // //---------------------------------------------------------------------------------------------------------------//"
END_VISUALIZATION
